// TIA Portal V20 export
FUNCTION "PMC_Config_Map02" : Void   // FC102, LAD
// stored: Namespace CITI_Logic, SetENOAutomatically false
BEGIN

REGION Network 1: Use Remote Configuration Values
   // <@TODO>
   // ################################################################
   // # Use SET and RESET instructions to Manually Configure the Memory Map.
   // #SEE CITI ENGINEER FOR CORRECT VALUES
   // # IF REMOTE CONFIGURATION IS DISABLED THEN THE CONFIGURATION BELOW WILL BE USED
   // # IF REMOTE CONFIGURATION IS EABLED THEN THE CONFIGURATION FROM JARVIS WILL BE USED (NOT A CURRENT OPTION)
   // ################################################################
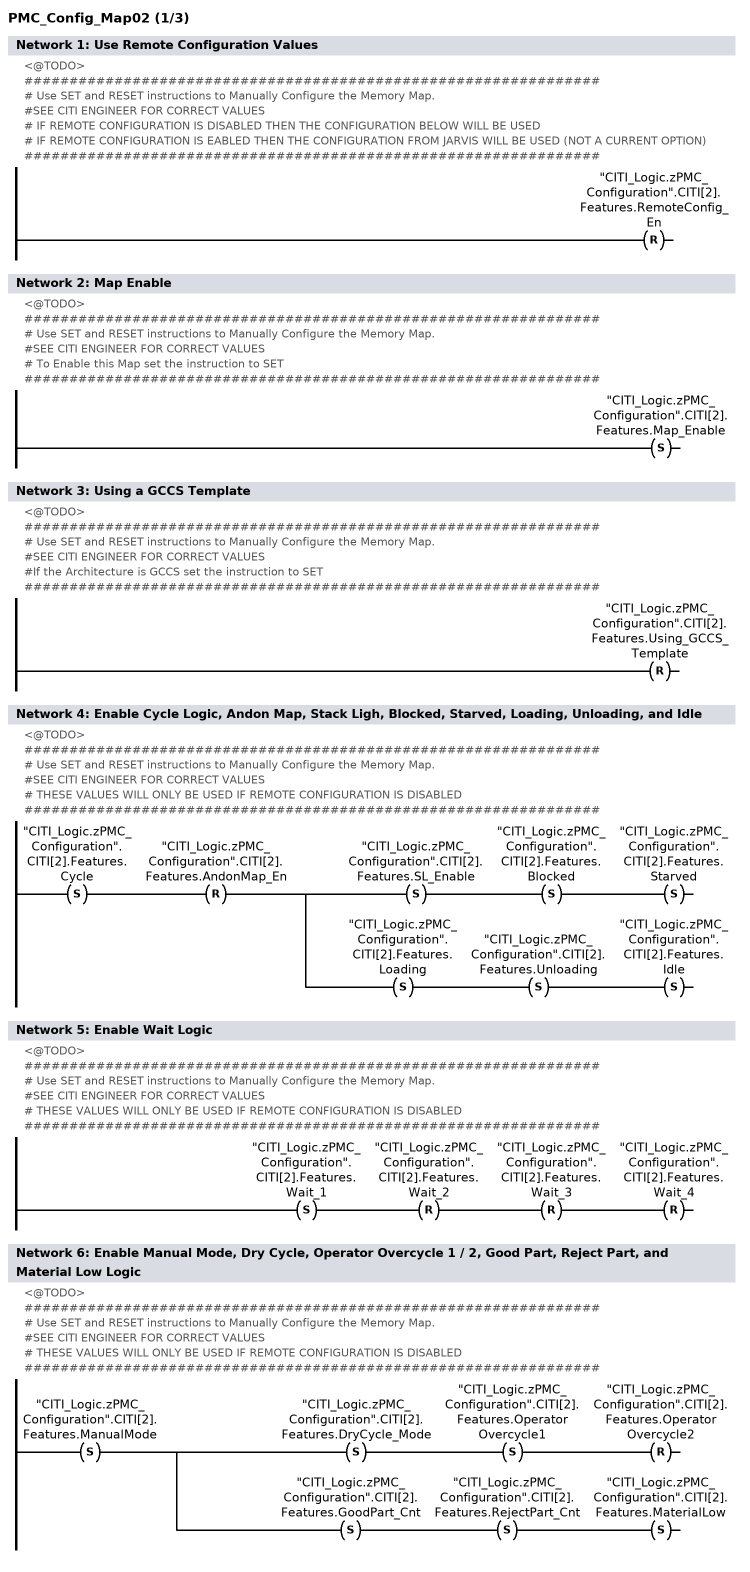
   RUNG wire#powerrail
      R_Coil( "CITI_Logic.zPMC_Configuration".CITI[2].Features.RemoteConfig_En )
   END_RUNG
   // the same network as SCL:
   "CITI_Logic.zPMC_Configuration".CITI[2].Features.RemoteConfig_En := FALSE;
END_REGION

REGION Network 2: Map Enable
   // <@TODO>
   // ################################################################
   // # Use SET and RESET instructions to Manually Configure the Memory Map.
   // #SEE CITI ENGINEER FOR CORRECT VALUES
   // # To Enable this Map set the instruction to SET
   // ################################################################
   RUNG wire#powerrail
      S_Coil( "CITI_Logic.zPMC_Configuration".CITI[2].Features.Map_Enable )
   END_RUNG
   // the same network as SCL:
   "CITI_Logic.zPMC_Configuration".CITI[2].Features.Map_Enable := TRUE;
END_REGION

REGION Network 3: Using a GCCS Template
   // <@TODO>
   // ################################################################
   // # Use SET and RESET instructions to Manually Configure the Memory Map.
   // #SEE CITI ENGINEER FOR CORRECT VALUES
   // #If the Architecture is GCCS set the instruction to SET
   // ################################################################
   RUNG wire#powerrail
      R_Coil( "CITI_Logic.zPMC_Configuration".CITI[2].Features.Using_GCCS_Template )
   END_RUNG
   // the same network as SCL:
   "CITI_Logic.zPMC_Configuration".CITI[2].Features.Using_GCCS_Template := FALSE;
END_REGION

REGION Network 4: Enable Cycle Logic, Andon Map, Stack Ligh, Blocked, Starved, Loading, Unloading, and Idle
   // <@TODO>
   // ################################################################
   // # Use SET and RESET instructions to Manually Configure the Memory Map.
   // #SEE CITI ENGINEER FOR CORRECT VALUES
   // # THESE VALUES WILL ONLY BE USED IF REMOTE CONFIGURATION IS DISABLED
   // ################################################################
   RUNG wire#powerrail
      S_Coil( "CITI_Logic.zPMC_Configuration".CITI[2].Features.Cycle )
      R_Coil( "CITI_Logic.zPMC_Configuration".CITI[2].Features.AndonMap_En )
      wire#w1
      S_Coil( "CITI_Logic.zPMC_Configuration".CITI[2].Features.SL_Enable )
      S_Coil( "CITI_Logic.zPMC_Configuration".CITI[2].Features.Blocked )
      S_Coil( "CITI_Logic.zPMC_Configuration".CITI[2].Features.Starved )
   END_RUNG
   RUNG wire#w1
      S_Coil( "CITI_Logic.zPMC_Configuration".CITI[2].Features.Loading )
      S_Coil( "CITI_Logic.zPMC_Configuration".CITI[2].Features.Unloading )
      S_Coil( "CITI_Logic.zPMC_Configuration".CITI[2].Features.Idle )
   END_RUNG
   // the same network as SCL:
   "CITI_Logic.zPMC_Configuration".CITI[2].Features.Cycle := TRUE;
   "CITI_Logic.zPMC_Configuration".CITI[2].Features.AndonMap_En := FALSE;
   "CITI_Logic.zPMC_Configuration".CITI[2].Features.SL_Enable := TRUE;
   "CITI_Logic.zPMC_Configuration".CITI[2].Features.Blocked := TRUE;
   "CITI_Logic.zPMC_Configuration".CITI[2].Features.Starved := TRUE;
   "CITI_Logic.zPMC_Configuration".CITI[2].Features.Loading := TRUE;
   "CITI_Logic.zPMC_Configuration".CITI[2].Features.Unloading := TRUE;
   "CITI_Logic.zPMC_Configuration".CITI[2].Features.Idle := TRUE;
END_REGION

REGION Network 5: Enable Wait Logic
   // <@TODO>
   // ################################################################
   // # Use SET and RESET instructions to Manually Configure the Memory Map.
   // #SEE CITI ENGINEER FOR CORRECT VALUES
   // # THESE VALUES WILL ONLY BE USED IF REMOTE CONFIGURATION IS DISABLED
   // ################################################################
   RUNG wire#powerrail
      S_Coil( "CITI_Logic.zPMC_Configuration".CITI[2].Features.Wait_1 )
      R_Coil( "CITI_Logic.zPMC_Configuration".CITI[2].Features.Wait_2 )
      R_Coil( "CITI_Logic.zPMC_Configuration".CITI[2].Features.Wait_3 )
      R_Coil( "CITI_Logic.zPMC_Configuration".CITI[2].Features.Wait_4 )
   END_RUNG
   // the same network as SCL:
   "CITI_Logic.zPMC_Configuration".CITI[2].Features.Wait_1 := TRUE;
   "CITI_Logic.zPMC_Configuration".CITI[2].Features.Wait_2 := FALSE;
   "CITI_Logic.zPMC_Configuration".CITI[2].Features.Wait_3 := FALSE;
   "CITI_Logic.zPMC_Configuration".CITI[2].Features.Wait_4 := FALSE;
END_REGION

REGION Network 6: Enable Manual Mode, Dry Cycle, Operator Overcycle 1 / 2, Good Part, Reject Part, and Material Low Logic
   // <@TODO>
   // ################################################################
   // # Use SET and RESET instructions to Manually Configure the Memory Map.
   // #SEE CITI ENGINEER FOR CORRECT VALUES
   // # THESE VALUES WILL ONLY BE USED IF REMOTE CONFIGURATION IS DISABLED
   // ################################################################
   RUNG wire#powerrail
      S_Coil( "CITI_Logic.zPMC_Configuration".CITI[2].Features.ManualMode )
      wire#w1
      S_Coil( "CITI_Logic.zPMC_Configuration".CITI[2].Features.DryCycle_Mode )
      S_Coil( "CITI_Logic.zPMC_Configuration".CITI[2].Features.OperatorOvercycle1 )
      R_Coil( "CITI_Logic.zPMC_Configuration".CITI[2].Features.OperatorOvercycle2 )
   END_RUNG
   RUNG wire#w1
      S_Coil( "CITI_Logic.zPMC_Configuration".CITI[2].Features.GoodPart_Cnt )
      S_Coil( "CITI_Logic.zPMC_Configuration".CITI[2].Features.RejectPart_Cnt )
      S_Coil( "CITI_Logic.zPMC_Configuration".CITI[2].Features.MaterialLow )
   END_RUNG
   // the same network as SCL:
   "CITI_Logic.zPMC_Configuration".CITI[2].Features.ManualMode := TRUE;
   "CITI_Logic.zPMC_Configuration".CITI[2].Features.DryCycle_Mode := TRUE;
   "CITI_Logic.zPMC_Configuration".CITI[2].Features.OperatorOvercycle1 := TRUE;
   "CITI_Logic.zPMC_Configuration".CITI[2].Features.OperatorOvercycle2 := FALSE;
   "CITI_Logic.zPMC_Configuration".CITI[2].Features.GoodPart_Cnt := TRUE;
   "CITI_Logic.zPMC_Configuration".CITI[2].Features.RejectPart_Cnt := TRUE;
   "CITI_Logic.zPMC_Configuration".CITI[2].Features.MaterialLow := TRUE;
END_REGION

REGION Network 7: Map Uses String Data, PUN, GM Part Number, Optional Data, Part Types, FTQ, and Andon Hold
   // <@TODO>
   // ################################################################
   // # Use SET and RESET instructions to Manually Configure the Memory Map.
   // #SEE CITI ENGINEER FOR CORRECT VALUES
   // # THESE VALUES WILL ONLY BE USED IF REMOTE CONFIGURATION IS DISABLED
   // ################################################################
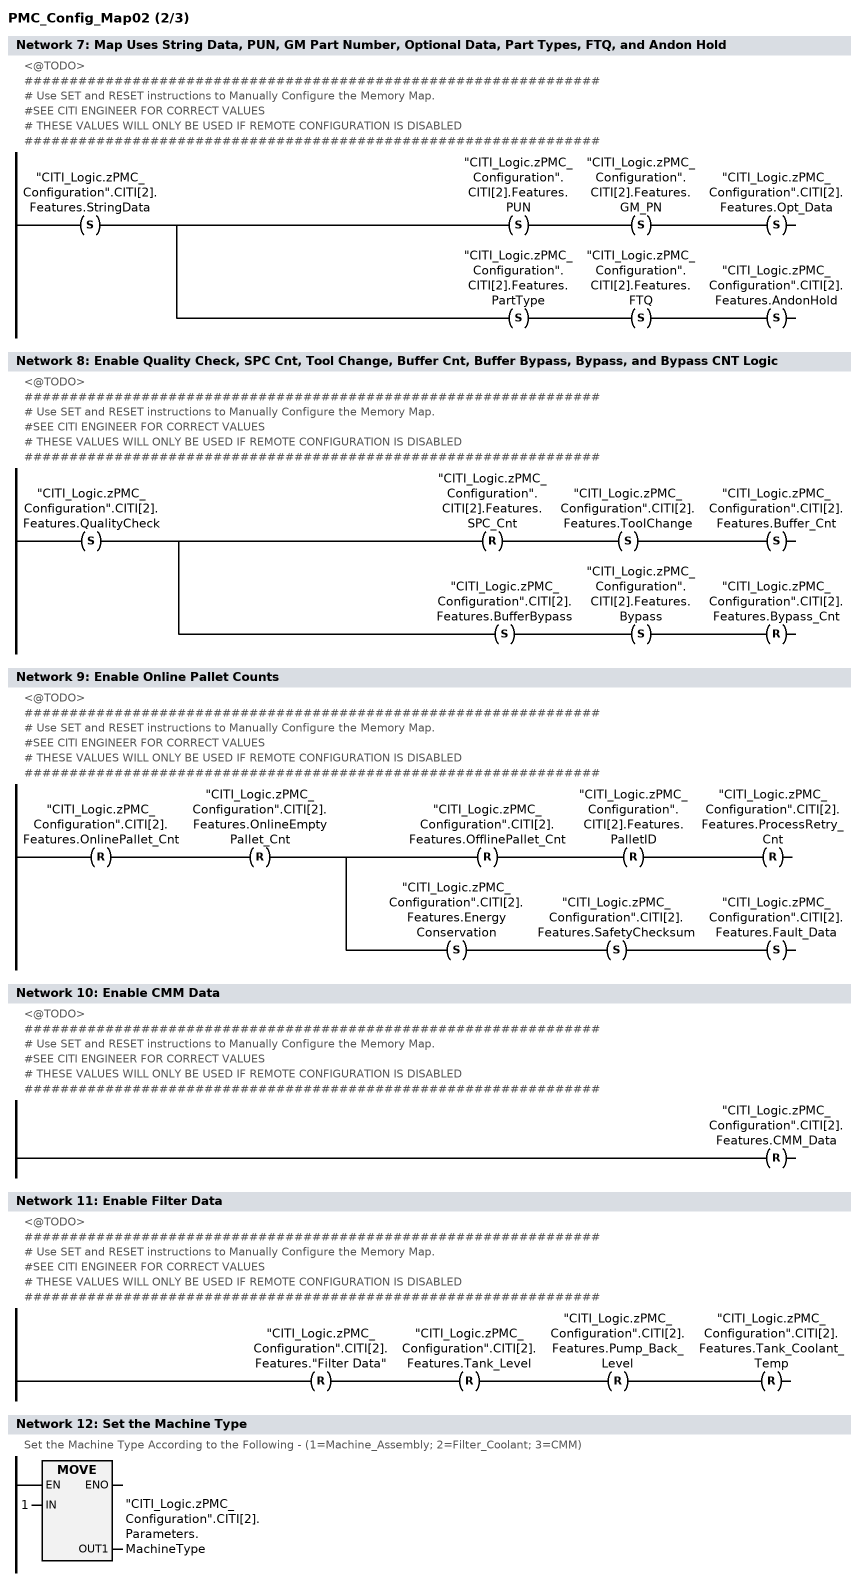
   RUNG wire#powerrail
      S_Coil( "CITI_Logic.zPMC_Configuration".CITI[2].Features.StringData )
      wire#w1
      S_Coil( "CITI_Logic.zPMC_Configuration".CITI[2].Features.PUN )
      S_Coil( "CITI_Logic.zPMC_Configuration".CITI[2].Features.GM_PN )
      S_Coil( "CITI_Logic.zPMC_Configuration".CITI[2].Features.Opt_Data )
   END_RUNG
   RUNG wire#w1
      S_Coil( "CITI_Logic.zPMC_Configuration".CITI[2].Features.PartType )
      S_Coil( "CITI_Logic.zPMC_Configuration".CITI[2].Features.FTQ )
      S_Coil( "CITI_Logic.zPMC_Configuration".CITI[2].Features.AndonHold )
   END_RUNG
   // the same network as SCL:
   "CITI_Logic.zPMC_Configuration".CITI[2].Features.StringData := TRUE;
   "CITI_Logic.zPMC_Configuration".CITI[2].Features.PUN := TRUE;
   "CITI_Logic.zPMC_Configuration".CITI[2].Features.GM_PN := TRUE;
   "CITI_Logic.zPMC_Configuration".CITI[2].Features.Opt_Data := TRUE;
   "CITI_Logic.zPMC_Configuration".CITI[2].Features.PartType := TRUE;
   "CITI_Logic.zPMC_Configuration".CITI[2].Features.FTQ := TRUE;
   "CITI_Logic.zPMC_Configuration".CITI[2].Features.AndonHold := TRUE;
END_REGION

REGION Network 8: Enable Quality Check, SPC Cnt, Tool Change, Buffer Cnt, Buffer Bypass, Bypass, and Bypass CNT Logic
   // <@TODO>
   // ################################################################
   // # Use SET and RESET instructions to Manually Configure the Memory Map.
   // #SEE CITI ENGINEER FOR CORRECT VALUES
   // # THESE VALUES WILL ONLY BE USED IF REMOTE CONFIGURATION IS DISABLED
   // ################################################################
   RUNG wire#powerrail
      S_Coil( "CITI_Logic.zPMC_Configuration".CITI[2].Features.QualityCheck )
      wire#w1
      R_Coil( "CITI_Logic.zPMC_Configuration".CITI[2].Features.SPC_Cnt )
      S_Coil( "CITI_Logic.zPMC_Configuration".CITI[2].Features.ToolChange )
      S_Coil( "CITI_Logic.zPMC_Configuration".CITI[2].Features.Buffer_Cnt )
   END_RUNG
   RUNG wire#w1
      S_Coil( "CITI_Logic.zPMC_Configuration".CITI[2].Features.BufferBypass )
      S_Coil( "CITI_Logic.zPMC_Configuration".CITI[2].Features.Bypass )
      R_Coil( "CITI_Logic.zPMC_Configuration".CITI[2].Features.Bypass_Cnt )
   END_RUNG
   // the same network as SCL:
   "CITI_Logic.zPMC_Configuration".CITI[2].Features.QualityCheck := TRUE;
   "CITI_Logic.zPMC_Configuration".CITI[2].Features.SPC_Cnt := FALSE;
   "CITI_Logic.zPMC_Configuration".CITI[2].Features.ToolChange := TRUE;
   "CITI_Logic.zPMC_Configuration".CITI[2].Features.Buffer_Cnt := TRUE;
   "CITI_Logic.zPMC_Configuration".CITI[2].Features.BufferBypass := TRUE;
   "CITI_Logic.zPMC_Configuration".CITI[2].Features.Bypass := TRUE;
   "CITI_Logic.zPMC_Configuration".CITI[2].Features.Bypass_Cnt := FALSE;
END_REGION

REGION Network 9: Enable Online Pallet Counts
   // <@TODO>
   // ################################################################
   // # Use SET and RESET instructions to Manually Configure the Memory Map.
   // #SEE CITI ENGINEER FOR CORRECT VALUES
   // # THESE VALUES WILL ONLY BE USED IF REMOTE CONFIGURATION IS DISABLED
   // ################################################################
   RUNG wire#powerrail
      R_Coil( "CITI_Logic.zPMC_Configuration".CITI[2].Features.OnlinePallet_Cnt )
      R_Coil( "CITI_Logic.zPMC_Configuration".CITI[2].Features.OnlineEmptyPallet_Cnt )
      wire#w1
      R_Coil( "CITI_Logic.zPMC_Configuration".CITI[2].Features.OfflinePallet_Cnt )
      R_Coil( "CITI_Logic.zPMC_Configuration".CITI[2].Features.PalletID )
      R_Coil( "CITI_Logic.zPMC_Configuration".CITI[2].Features.ProcessRetry_Cnt )
   END_RUNG
   RUNG wire#w1
      S_Coil( "CITI_Logic.zPMC_Configuration".CITI[2].Features.EnergyConservation )
      S_Coil( "CITI_Logic.zPMC_Configuration".CITI[2].Features.SafetyChecksum )
      S_Coil( "CITI_Logic.zPMC_Configuration".CITI[2].Features.Fault_Data )
   END_RUNG
   // the same network as SCL:
   "CITI_Logic.zPMC_Configuration".CITI[2].Features.OnlinePallet_Cnt := FALSE;
   "CITI_Logic.zPMC_Configuration".CITI[2].Features.OnlineEmptyPallet_Cnt := FALSE;
   "CITI_Logic.zPMC_Configuration".CITI[2].Features.OfflinePallet_Cnt := FALSE;
   "CITI_Logic.zPMC_Configuration".CITI[2].Features.PalletID := FALSE;
   "CITI_Logic.zPMC_Configuration".CITI[2].Features.ProcessRetry_Cnt := FALSE;
   "CITI_Logic.zPMC_Configuration".CITI[2].Features.EnergyConservation := TRUE;
   "CITI_Logic.zPMC_Configuration".CITI[2].Features.SafetyChecksum := TRUE;
   "CITI_Logic.zPMC_Configuration".CITI[2].Features.Fault_Data := TRUE;
END_REGION

REGION Network 10: Enable CMM Data
   // <@TODO>
   // ################################################################
   // # Use SET and RESET instructions to Manually Configure the Memory Map.
   // #SEE CITI ENGINEER FOR CORRECT VALUES
   // # THESE VALUES WILL ONLY BE USED IF REMOTE CONFIGURATION IS DISABLED
   // ################################################################
   RUNG wire#powerrail
      R_Coil( "CITI_Logic.zPMC_Configuration".CITI[2].Features.CMM_Data )
   END_RUNG
   // the same network as SCL:
   "CITI_Logic.zPMC_Configuration".CITI[2].Features.CMM_Data := FALSE;
END_REGION

REGION Network 11: Enable Filter Data
   // <@TODO>
   // ################################################################
   // # Use SET and RESET instructions to Manually Configure the Memory Map.
   // #SEE CITI ENGINEER FOR CORRECT VALUES
   // # THESE VALUES WILL ONLY BE USED IF REMOTE CONFIGURATION IS DISABLED
   // ################################################################
   RUNG wire#powerrail
      R_Coil( "CITI_Logic.zPMC_Configuration".CITI[2].Features."Filter Data" )
      R_Coil( "CITI_Logic.zPMC_Configuration".CITI[2].Features.Tank_Level )
      R_Coil( "CITI_Logic.zPMC_Configuration".CITI[2].Features.Pump_Back_Level )
      R_Coil( "CITI_Logic.zPMC_Configuration".CITI[2].Features.Tank_Coolant_Temp )
   END_RUNG
   // the same network as SCL:
   "CITI_Logic.zPMC_Configuration".CITI[2].Features."Filter Data" := FALSE;
   "CITI_Logic.zPMC_Configuration".CITI[2].Features.Tank_Level := FALSE;
   "CITI_Logic.zPMC_Configuration".CITI[2].Features.Pump_Back_Level := FALSE;
   "CITI_Logic.zPMC_Configuration".CITI[2].Features.Tank_Coolant_Temp := FALSE;
END_REGION

REGION Network 12: Set the Machine Type
   // Set the Machine Type According to the Following - (1=Machine_Assembly; 2=Filter_Coolant; 3=CMM)
   RUNG wire#powerrail
      Move(in := 1, out1 => "CITI_Logic.zPMC_Configuration".CITI[2].Parameters.MachineType)
   END_RUNG
   // the same network as SCL:
   "CITI_Logic.zPMC_Configuration".CITI[2].Parameters.MachineType := 1;
END_REGION

REGION Network 13: CITI Parameters
   // <@TODO>
   // ################################################################
   // #SEE CITI ENGINEER FOR CORRECT VALUES
   // # THESE VALUES WILL ONLY BE USED IF REMOTE CONFIGURATION IS DISABLED
   // ################################################################
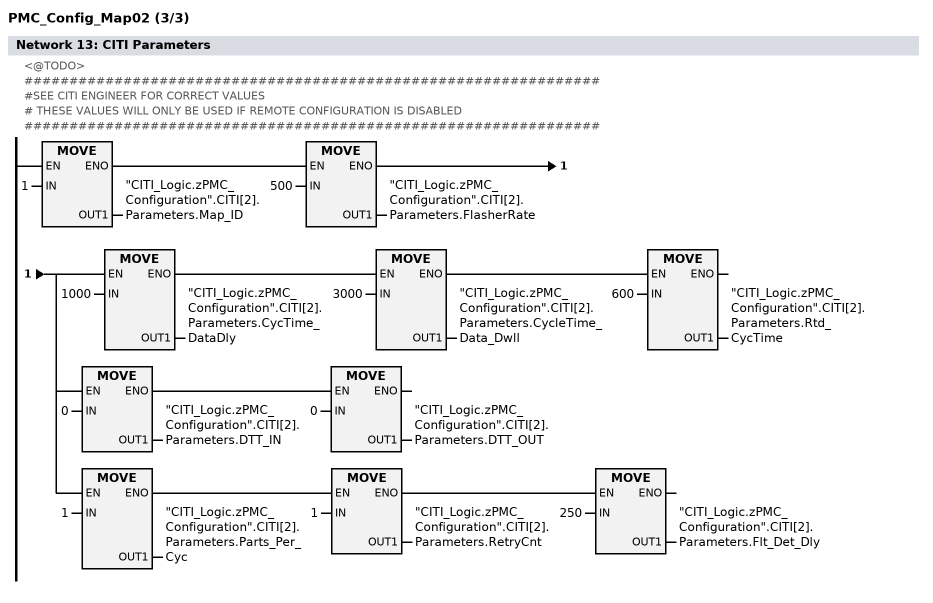
   RUNG wire#powerrail
      Move(in := 1, out1 => "CITI_Logic.zPMC_Configuration".CITI[2].Parameters.Map_ID)
      Move(in := 500, out1 => "CITI_Logic.zPMC_Configuration".CITI[2].Parameters.FlasherRate)
      wire#w1
      Move(in := 1000, out1 => "CITI_Logic.zPMC_Configuration".CITI[2].Parameters.CycTime_DataDly)
      Move(in := 3000, out1 => "CITI_Logic.zPMC_Configuration".CITI[2].Parameters.CycleTime_Data_Dwll)
      Move(in := 600, out1 => "CITI_Logic.zPMC_Configuration".CITI[2].Parameters.Rtd_CycTime)
   END_RUNG
   RUNG wire#w1
      Move(in := 0, out1 => "CITI_Logic.zPMC_Configuration".CITI[2].Parameters.DTT_IN)
      Move(in := 0, out1 => "CITI_Logic.zPMC_Configuration".CITI[2].Parameters.DTT_OUT)
   END_RUNG
   RUNG wire#w1
      Move(in := 1, out1 => "CITI_Logic.zPMC_Configuration".CITI[2].Parameters.Parts_Per_Cyc)
      Move(in := 1, out1 => "CITI_Logic.zPMC_Configuration".CITI[2].Parameters.RetryCnt)
      Move(in := 250, out1 => "CITI_Logic.zPMC_Configuration".CITI[2].Parameters.Flt_Det_Dly)
   END_RUNG
   // the same network as SCL:
   "CITI_Logic.zPMC_Configuration".CITI[2].Parameters.Map_ID := 1;
   "CITI_Logic.zPMC_Configuration".CITI[2].Parameters.FlasherRate := 500;
   "CITI_Logic.zPMC_Configuration".CITI[2].Parameters.CycTime_DataDly := 1000;
   "CITI_Logic.zPMC_Configuration".CITI[2].Parameters.CycleTime_Data_Dwll := 3000;
   "CITI_Logic.zPMC_Configuration".CITI[2].Parameters.Rtd_CycTime := 600;
   "CITI_Logic.zPMC_Configuration".CITI[2].Parameters.DTT_IN := 0;
   "CITI_Logic.zPMC_Configuration".CITI[2].Parameters.DTT_OUT := 0;
   "CITI_Logic.zPMC_Configuration".CITI[2].Parameters.Parts_Per_Cyc := 1;
   "CITI_Logic.zPMC_Configuration".CITI[2].Parameters.RetryCnt := 1;
   "CITI_Logic.zPMC_Configuration".CITI[2].Parameters.Flt_Det_Dly := 250;
END_REGION
END_FUNCTION
